FUNCTION_BLOCK NullError_TestSuite EXTENDS TcUnit.FB_TestSuite

TestErrorType();
TestMessage();

METHOD PUBLIC TestErrorType
VAR
	error : NullError;
END_VAR
TEST('TestErrorType');

AssertEquals_String(
	Actual := error.ErrorType,
	Expected := '',
	Message := 'Did not return the expected ErrorType'
);

TEST_FINISHED();
END_METHOD

METHOD PUBLIC TestMessage
VAR
	error : NullError;
END_VAR
TEST('TestMessage');

AssertEquals_String(
	Actual := error.Message,
	Expected := '',
	Message := 'Did not return the expected Message'
);

TEST_FINISHED();
END_METHOD

END_FUNCTION_BLOCK

(* stored: Version 1.1.0.1, ProductVersion 3.1.4024.12
   POU NullError_TestSuite: Id {b1cc6e12-fdb1-4945-b863-3dcc1e456d61}, SpecialFunc None
   Method TestErrorType: Id {ce53f6c0-86dd-4bff-9bc5-d7a9429a3eac}
   Method TestMessage: Id {7726e46b-57d9-4b17-ba41-e98819a67da6} *)
